RoboDK station: CSU Expo Station.rdk

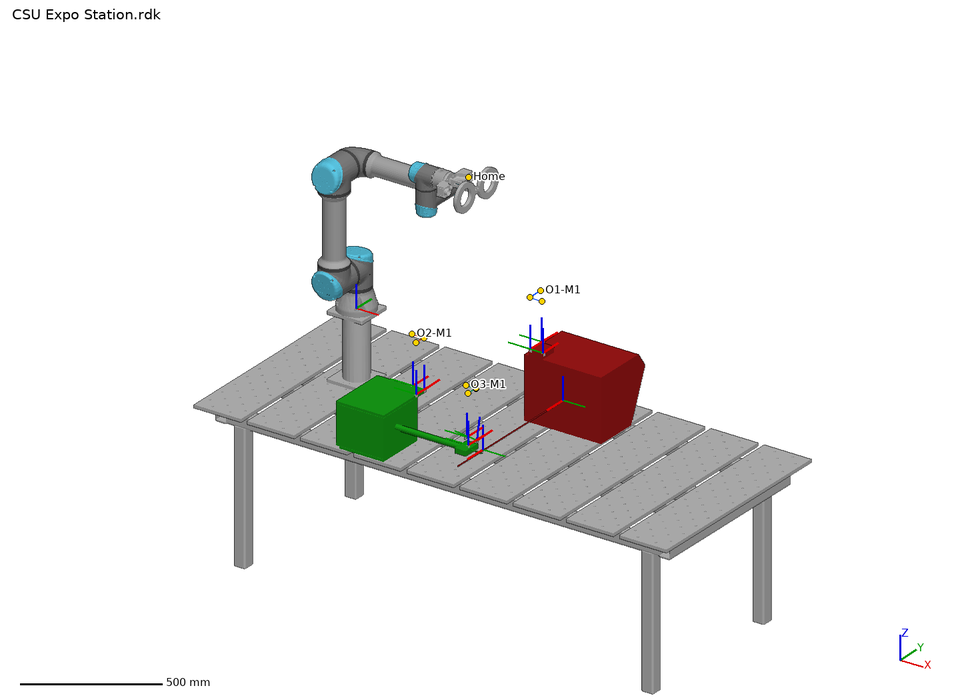
[picture v0: the station drawn from its stored meshes, robots at their saved joint values, targets as dots, program paths as lines]
Station CSU Expo Station (saved by RoboDK 5.0.1). Poses are relative to the parent item; angles as X-Y-Z fixed-axis rotations.
  - object Welding Table at (-1600, 2170, 0) mm, rotated rx 90 ry 0 rz 0 deg, size 2032 x 628.6 x 889 mm, geometry from Welding Table.STEP
  - object Tower_V4.1 (2) at (-1504.7, 555.63, 733.6) mm, size 152.4 x 152.4 x 279.4 mm, geometry from Tower_V4.1 (2).STEP
  - object X-Ray Box (3) at (-679.2, 641.63, 724.08) mm, rotated rx 0 ry 0 rz -90 deg, size 914.8 x 330 x 284 mm, geometry from X-Ray Box (3).STEP
  - object Kappa Expo (1) at (-1059.7, 166.63, 724.08) mm, rotated rx 0 ry 0 rz -90 deg, size 256 x 575.5 x 181.2 mm, geometry from Kappa Expo (1).STEP
  - frame UR5e Base at (-1504.7, 555.63, 1013) mm
    - robot UR5e: 6 axes, payload 5 kg, reach 850 mm, repeatability 0.03 mm, weight 18.4 kg
        modified DH rows (alpha deg, a mm, theta deg, d mm): 0, 0, 0, 162.5; 90, 0, 180, 0; 0, 425, 0, 0; 0, 392.25, 0, 133.3; -90, 0, 0, 99.7; 90, 0, 180, 99.6
        joint limits [-360, -360, -360, -360, -360, -360] to [360, 360, 360, 360, 360, 360]; home [0, -90, -90, 0, 90, 0]; saved at [0, -90, -90, 0, 90, 0]
      - tool Left Camera, TCP at (-69.39, 0, 34.3) mm, size 256 x 114.2 x 122.3 mm
      - tool Right Camera, TCP at (69.39, 0, 34.3) mm
    - target Home (Cartesian target) at (526.15, -63.91, 687.2) mm, rotated rx -90 ry 0 rz -90 deg; joints [0, -90, -90, 0, 90, 0] of UR5e
    - target O1-M1 (Cartesian target) at (682, 157, 198.5) mm, rotated rx 180 ry 0 rz -90 deg; joints [18.498, -122.802, -85.726, -61.472, 90.002, 18.498] of UR5e
    - target O1-M2 (Cartesian target) at (682, 89, 198.5) mm, rotated rx -180 ry 0 rz -90 deg; joints [12.914, -122.158, -86.796, -61.046, 89.997, 12.914] of UR5e
    - target O1-M3 (Cartesian target) at (735, 89, 198.5) mm, rotated rx 180 ry 0 rz -90 deg; joints [11.974, -128.74, -75.588, -65.672, 89.998, 11.974] of UR5e
    - target O2-M1 (Cartesian target) at (392, -217.96, 96) mm, rotated rx 180 ry 0 rz -90 deg; joints [-20.326, -111.217, -125.737, -33.048, 90.003, -20.326] of UR5e
    - target O2-M2 (Cartesian target) at (442, -217.96, 96) mm, rotated rx 180 ry 0 rz -90 deg; joints [-18.383, -115.073, -118.98, -35.949, 90, -18.383] of UR5e
    - target O2-M3 (Cartesian target) at (442, -267.96, 96) mm, rotated rx 180 ry 0 rz -90 deg; joints [-23.481, -117.773, -114.117, -38.113, 89.999, -23.481] of UR5e
    - target O3-M1 (Cartesian target) at (723, -359.5, 44.31) mm, rotated rx 180 ry 0 rz -90 deg; joints [-21.553, -153.256, -53.33, -63.416, 90, -21.553] of UR5e
    - target O3-M2 (Cartesian target) at (765, -359.5, 44.31) mm, rotated rx 180 ry 0 rz -90 deg; joints [-20.535, -159.517, -40.305, -70.18, 90.001, -20.535] of UR5e
    - target O3-M3 (Cartesian target) at (765, -409.5, 44.31) mm, rotated rx 180 ry 0 rz -90 deg; joints [-23.553, -165.459, -27.955, -76.587, 90.001, -23.553] of UR5e
    - target Target 11 (Cartesian target) at (765.02, -359.5, 46.15) mm, rotated rx -180 ry 0 rz -89.99 deg; joints [-20.534, -159.392, -40.279, -70.329, 90.004, -20.543] of UR5e
  - Python program Prog1 (listed below)
  - program OB1 (6 instructions, listed below)
  - program OB2 (6 instructions, listed below)
  - program OB3 (6 instructions, listed below)
  - program hOME (4 instructions, listed below)
  - Python program Prog6 (listed below)
  - frame Specimen at (-689.2, 166.63, 844.08) mm, rotated rx 0 ry 0 rz -90 deg
  - frame O1-M1 at (-819.7, 715.63, 1010.08) mm, rotated rx 0 ry 0 rz 90 deg
    - object O1-M1 at (3, -3, 0) mm, rotated rx 0 ry 0 rz 90 deg, size 10 x 10 x 10 mm, geometry from Fiducial Edge (1).STEP
  - frame O1-M2 at (-819.7, 644.63, 1010.08) mm, rotated rx 0 ry 0 rz 90 deg
    - object O1-M2 at (0, -3, 0) mm, rotated rx 0 ry 0 rz 90 deg, size 10 x 10 x 10 mm, geometry from Fiducal Corner.STEP
  - frame O1-M3 at (-766.7, 644.63, 1010.08) mm, rotated rx 0 ry 0 rz 90 deg
    - object O1-M3 at (0, -3, 0) mm, rotated rx 0 ry 0 rz -90 deg, size 10 x 10 x 10 mm, geometry from Fiducial Edge (1).STEP
  - frame O2-M1 at (-1109.7, 337.67, 907.33) mm, rotated rx 0 ry 0 rz 90 deg
    - object O2-M1 at (0, 3, 0) mm, size 10 x 10 x 10 mm, geometry from Fiducial Edge (1).STEP
  - frame O2-M2 at (-1059.7, 337.67, 907.33) mm, rotated rx 0 ry 0 rz 90 deg
    - object O2-M2 at (0, 3, 0) mm, rotated rx 0 ry 0 rz -180 deg, size 10 x 10 x 10 mm, geometry from Fiducal Corner.STEP
  - frame O2-M3 at (-1059.7, 287.67, 907.33) mm, rotated rx 0 ry 0 rz 90 deg
    - object O2-M3 at (0, 3, 0) mm, rotated rx 0 ry 0 rz -90 deg, size 10 x 10 x 10 mm, geometry from Fiducial Edge (1).STEP
  - frame O3-M1 at (-778.7, 196.13, 856.08) mm, rotated rx 0 ry 0 rz 90 deg
    - object O3-M1 at (0, 3, 0) mm, rotated rx 0 ry 0 rz 90 deg, size 10 x 10 x 10 mm, geometry from Fiducial Edge (1).STEP
  - frame O3-M2 at (-735.04, 196.13, 855.98) mm, rotated rx 6.36 ry -0.02 rz 90.28 deg
    - object O3-M2 at (0, 3, 0) mm, rotated rx 0 ry 0 rz -180 deg, size 10 x 10 x 10 mm, geometry from Fiducal Corner.STEP
  - frame O3-M3 at (-736.7, 146.13, 856.08) mm, rotated rx 0 ry 0 rz 90 deg
    - object O3-M3 at (0, 3, 0) mm, rotated rx 0 ry 0 rz -90 deg, size 10 x 10 x 10 mm, geometry from Fiducial Edge (1).STEP
  - frame X-Ray Outlet at (-679.2, 642.63, 849.08) mm, rotated rx 0 ry 0 rz -90 deg
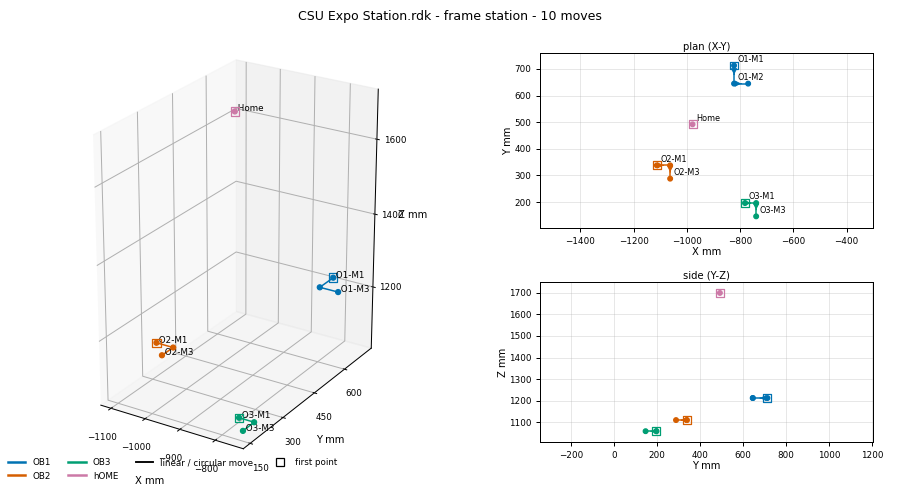
[picture p0: tool path of CSU Expo Station.rdk in frame station, 10 of 10 moves have a stored position in this frame; points joined in program order, loops and branches not executed]

--- Python program Prog1 ---
from robolink import *    # RoboDK's API
from robodk import *      # Math toolbox for robots
import logging
import sys, time, math

RDK = robolink.Robolink()

# OpenCV is an open source Computer Vision toolkit, which you can use to filter and analyse images
robolink.import_install('cv2', 'opencv-contrib-python', RDK)
robolink.import_install('numpy', RDK)

sys.path.insert(1, r'C:\Users\PoThe\OneDrive\Desktop\VimbaPython_Source')
import numpy as np
import cv2 as cv
import cv2
from cv2 import VideoCapture, aruco
from vimba import *
import measure_class

logging.basicConfig(filename="TestRun.log",level=logging.INFO,filemode='w')

calib_path  = r'C:\Users\PoThe\OneDrive\Desktop\VimbaPython_Source'
camera_matrix   = np.loadtxt(calib_path+'\cameraMatrix.txt', delimiter=',')
camera_distortion   = np.loadtxt(calib_path+'\cameraDistortion.txt', delimiter=',')

marker_actual = 6 #[mm]

marker_size  =  marker_actual/10 # how it will be processed [cm]

# Define Robot:
robot = RDK.Item('UR5e', ITEM_TYPE_ROBOT)
O1M1 = RDK.Item('O1-M1',ITEM_TYPE_OBJECT)

O1_M1_xyz = list()

O1_M1 = measure_class.measure(0,0,0,0)
O1M1_Xray = (73, -140.5, 161.00)
def offset(y,z):
    osy = y+30
    osz = z+6
    return osy, osz

TCP = robot.Pose()
O1_M1.measuring(marker_size, calib_path, camera_matrix, camera_distortion)
cv2.destroyAllWindows()
x = -O1_M1.x
O1_M1_xyz.append(x)
O1_M1_xyz.append(O1_M1.y)
O1_M1_xyz.append(O1_M1.z)

O1M1_Base = TCP*transl(O1_M1_xyz)
x,y,z,rx,ry,rz = Pose_2_TxyzRxyz(O1M1_Base)
y,z = offset(y,z)
O1M1_Base = TxyzRxyz_2_Pose([x,y,z,rx,ry,rz])

O1_X1 = O1M1_Base*transl(O1M1_Xray)
x1,y1,z1,rx1,ry1,rz1 = Pose_2_TxyzRxyz(O1_X1)

logging.info("Marker 1 to base: %s", O1M1_Base)

logging.info("X-ray to base: %s", O1_X1)

--- program OB1 (robot UR5e) ---
  Set Ref.: UR5e Base
  Set Tool: Left Camera
  Set speed (200.0 mm/s)
  MoveL (O1-M1)
  MoveL (O1-M2)
  MoveL (O1-M3)

--- program OB2 (robot UR5e) ---
  Set Ref.: UR5e Base
  Set Tool: Left Camera
  Set speed (200.0 mm/s)
  MoveL (O2-M1)
  MoveL (O2-M2)
  MoveL (O2-M3)

--- program OB3 (robot UR5e) ---
  Set Ref.: UR5e Base
  Set Tool: Left Camera
  Set speed (200.0 mm/s)
  MoveL (O3-M1)
  MoveL (O3-M2)
  MoveL (O3-M3)

--- program hOME (robot UR5e) ---
  Set Ref.: UR5e Base
  Set Tool: Left Camera
  Set speed (100.0 mm/s)
  MoveL (Home)

--- Python program Prog6 ---
from robolink import *    # RoboDK's API
from robodk import *      # Math toolbox for robots
import logging
import sys, time, math

RDK = robolink.Robolink()

# OpenCV is an open source Computer Vision toolkit, which you can use to filter and analyse images
robolink.import_install('cv2', 'opencv-contrib-python', RDK)
robolink.import_install('numpy', RDK)

sys.path.insert(1, r'C:\Users\PoThe\OneDrive\Desktop\VimbaPython_Source')
import numpy as np
import cv2 as cv
import cv2
from cv2 import VideoCapture, aruco
from vimba import *
import measure_class

logging.basicConfig(filename="TestRun.log",level=logging.INFO,filemode='w')

calib_path  = r'C:\Users\PoThe\OneDrive\Desktop\VimbaPython_Source'
camera_matrix   = np.loadtxt(calib_path+'\cameraMatrix.txt', delimiter=',')
camera_distortion   = np.loadtxt(calib_path+'\cameraDistortion.txt', delimiter=',')

marker_actual = 6 #[mm]

marker_size  =  marker_actual/10 # how it will be processed [cm]

# Program example:
robot = RDK.Item('UR5e', ITEM_TYPE_ROBOT)
Home = RDK.Item('Home', ITEM_TYPE_TARGET)
O1M1 = RDK.Item('O1-M1', ITEM_TYPE_TARGET)
O1M2 = RDK.Item('O1-M2', ITEM_TYPE_TARGET)
O1M3 = RDK.Item('O1-M3', ITEM_TYPE_TARGET)
O2M1 = RDK.Item('O2-M1', ITEM_TYPE_TARGET)
O2M2 = RDK.Item('O2-M2', ITEM_TYPE_TARGET)
O2M3 = RDK.Item('O2-M3', ITEM_TYPE_TARGET)
O3M1 = RDK.Item('O3-M1', ITEM_TYPE_TARGET)
O3M2 = RDK.Item('O3-M2', ITEM_TYPE_TARGET)
O3M3 = RDK.Item('O3-M3', ITEM_TYPE_TARGET)

#ArUco Markers
O1_M1 = measure_class.measure(0,0,0,0)
O1_M2 = measure_class.measure(0,0,0,0)
O1_M3 = measure_class.measure(0,0,0,0)
O2_M1 = measure_class.measure(0,0,0,0)
O2_M2 = measure_class.measure(0,0,0,0)
O2_M3 = measure_class.measure(0,0,0,0)
O3_M1 = measure_class.measure(0,0,0,0)
O3_M2 = measure_class.measure(0,0,0,0)
O3_M3 = measure_class.measure(0,0,0,0)

#xyz coordinates
O1_M1_xyz = list()
O1_M2_xyz = list()
O1_M3_xyz = list()
O2_M1_xyz = list()
O2_M2_xyz = list()
O2_M3_xyz = list()
O3_M1_xyz = list()
O3_M2_xyz = list()
O3_M3_xyz = list()

#xyz of the reference frame 'X-ray Output' with respect to marker locations
#O1M1_Xray = (140.5, -71.00, -161.00)
O1M1_Xray = (73, -140.5, 161.00)
O1M2_Xray = (-2, -140.5, 161.00)
O1M3_Xray = (-2, -87.500, 161.00)

O2M1_Xray = (-304.960, -433.500, 58.250)
O2M2_Xray = (-304.960, -383.500, 58.250)
O2M3_Xray = (-354.960, -383.500, 58.250)

#xyz of the reference frame 'Specimen' with respect to marker locations
O3M1_Spec = (-29.5, -89.500, 12.000)
O3M2_Spec = (-29.504, -45.838, 11.908)
O3M3_Spec = (-20.500, -47.50, 12.00)

XR_xlist = list()
XR_ylist = list()
XR_zlist = list()
S_xlist = list()
S_ylist = list()
S_zlist = list()

def offset(y,z):
    osy = y+30
    osz = z+6
    return osy, osz

def home():
    robot.MoveL(Home)

def object1():

#MARKER 1
    #--------------------------------------------------------------------------------------------------------------------
    robot.MoveL(O1M1)
    TCP = robot.Pose()
    O1_M1.measuring(marker_size, calib_path, camera_matrix, camera_distortion)
    cv2.destroyAllWindows()
    x = -O1_M1.x
    O1_M1_xyz.append(x)
    O1_M1_xyz.append(O1_M1.y)
    O1_M1_xyz.append(O1_M1.z)

    O1M1_Base = TCP*transl(O1_M1_xyz)
    x,y,z,rx,ry,rz = Pose_2_TxyzRxyz(O1M1_Base)
    y,z = offset(y,z)
    O1M1_Base = TxyzRxyz_2_Pose([x,y,z,rx,ry,rz])

    O1_X1 = O1M1_Base*transl(O1M1_Xray)
    x1,y1,z1,rx1,ry1,rz1 = Pose_2_TxyzRxyz(O1_X1)
    XR_xlist.append(x1)
    XR_ylist.append(y1)
    XR_zlist.append(z1)
    logging.info("Marker 1 to base: %s", O1M1_Base)
    #--------------------------------------------------------------------------------------------------------------------

#MARKER 2
    #--------------------------------------------------------------------------------------------------------------------
    robot.MoveL(O1M2)
    TCP = robot.Pose()
    O1_M2.measuring(marker_size, calib_path, camera_matrix, camera_distortion)
    cv2.destroyAllWindows()
    x = -O1_M2.x
    O1_M2_xyz.append(x)
    O1_M2_xyz.append(O1_M2.y)
    O1_M2_xyz.append(O1_M2.z)

    O1M2_Base = TCP*transl(O1_M2_xyz)
    x,y,z,rx,ry,rz = Pose_2_TxyzRxyz(O1M2_Base)
    y,z = offset(y,z)
    O1M2_Base = TxyzRxyz_2_Pose([x,y,z,rx,ry,rz])

    O1_X2 = O1M2_Base*transl(O1M2_Xray)
    x2,y2,z2,rx2,ry2,rz2 = Pose_2_TxyzRxyz(O1_X2)
    XR_xlist.append(x2)
    XR_ylist.append(y2)
    XR_zlist.append(z2)
    logging.info("Marker 2 to base: %s", O1M2_Base)
    #--------------------------------------------------------------------------------------------------------------------

#MARKER 3
    #--------------------------------------------------------------------------------------------------------------------
    robot.MoveL(O1M3)
    TCP = robot.Pose()
    O1_M3.measuring(marker_size, calib_path, camera_matrix, camera_distortion)
    cv2.destroyAllWindows()
    x = -O1_M3.x
    O1_M3_xyz.append(x)
    O1_M3_xyz.append(O1_M3.y)
    O1_M3_xyz.append(O1_M3.z)

    O1M3_Base = TCP*transl(O1_M3_xyz)
    #logging.info("Marker ID: %s \nCamera Pos w/ respect to marker: x = %2.3f, y = %2.3f, z = %2.3f \nMarker matrix w/respect to base: %s\n", O1_M3.markerid[0], O1_M3.x, O1_M3.y, O1_M3.z, O1M3_Base)
    x,y,z,rx,ry,rz = Pose_2_TxyzRxyz(O1M3_Base)
    y,z = offset(y,z)
    O1M3_Base = TxyzRxyz_2_Pose([x,y,z,rx,ry,rz])
    logging.info("Marker 3 to base: %s", O1M3_Base)

    O1_X3 = O1M3_Base*transl(O1M3_Xray)
    x3,y3,z3,rx3,ry3,rz3 = Pose_2_TxyzRxyz(O1_X3)
    XR_xlist.append(x3)
    XR_ylist.append(y3)
    XR_zlist.append(z3)
    #--------------------------------------------------------------------------------------------------------------------

    logging.info("X-ray coordinates with respect to Base: \nPosition 1: %s \nPosition 2: %s \nPosition 3: %s",O1_X1, O1_X2, O1_X3)

def object2():
#MARKER 4
    #------------------------------------------------------------------------------------------------------------------
    robot.MoveL(O2M1)
    TCP = robot.Pose()
    O2_M1.measuring(marker_size, calib_path, camera_matrix, camera_distortion)
    cv2.destroyAllWindows()
    x = -O2_M1.x
    O2_M1_xyz.append(x)
    O2_M1_xyz.append(O2_M1.y)
    O2_M1_xyz.append(O2_M1.z)
    O2M1_Base = TCP*transl(O2_M1_xyz)

    O2M1_Base = TCP*transl(O2_M1_xyz)
    x,y,z,rx,ry,rz = Pose_2_TxyzRxyz(O2M1_Base)
    #y,z = offset(y,z)
    O2M1_Base = TxyzRxyz_2_Pose([x,y,z,rx,ry,rz])


    O2_X1 = O2M1_Base*transl(O2M1_Xray)
    x4,y4,z4,rx4,ry4,rz4 = Pose_2_TxyzRxyz(O2_X1)
    XR_xlist.append(x4)
    XR_ylist.append(y4)
    XR_zlist.append(z4)
    logging.info("Marker 4 with respect to base: %s", O2M1_Base)

#MARKER 5
    #----------------------------------------------------------------------------------------------------------------------
    robot.MoveL(O2M2)
    TCP = robot.Pose()
    O2_M2.measuring(marker_size, calib_path, camera_matrix, camera_distortion)
    cv2.destroyAllWindows()
    x = -O2_M2.x
    O2_M2_xyz.append(x)
    O2_M2_xyz.append(O2_M2.y)
    O2_M2_xyz.append(O2_M2.z)
    O2M2_Base = TCP*transl(O2_M2_xyz)

    O2M2_Base = TCP*transl(O2_M2_xyz)
    x2,y2,z2,rx2,ry2,rz2 = Pose_2_TxyzRxyz(O2M2_Base)
    #y2,z2 = offset(y2,z2)
    O2M2_Base = TxyzRxyz_2_Pose([x2,y2,z2,rx2,ry2,rz2])

    logging.info("Marker 5 with respect to base: %s", O2M2_Base)
    O2_X2 = O2M2_Base*transl(O2M2_Xray)
    x5,y5,z5,rx5,ry5,rz5 = Pose_2_TxyzRxyz(O2_X2)
    XR_xlist.append(x5)
    XR_ylist.append(y5)
    XR_zlist.append(z5)

    #-------------------------------------------------------------------------------------------------------------------------------

#MARKER 6
    #-----------------------------------------------------------------------------------------------------------------------------
    robot.MoveL(O2M3)
    TCP = robot.Pose()
    O2_M3.measuring(marker_size, calib_path, camera_matrix, camera_distortion)
    cv2.destroyAllWindows()

    x = -O2_M3.x
    O2_M3_xyz.append(x)
    O2_M3_xyz.append(O2_M3.y)
    O2_M3_xyz.append(O2_M3.z)
    O2M3_Base = TCP*transl(O2_M3_xyz)

    O2M3_Base = TCP*transl(O2_M3_xyz)
    x3,y3,z3,rx3,ry3,rz3 = Pose_2_TxyzRxyz(O2M3_Base)
    y3,z3 = offset(y3,z3)
    O2M3_Base = TxyzRxyz_2_Pose([x3,y3,z3,rx3,ry3,rz3])
    #logging.info("Marker with respect to base: %s",O2M3_Base)
    O2_X3 = O2M3_Base*transl(O2M3_Xray)
    x6,y6,z6,rx6,ry6,rz6 = Pose_2_TxyzRxyz(O2_X3)
    XR_xlist.append(x6)
    XR_ylist.append(y6)
    XR_zlist.append(z6)
    logging.info("Marker 6 with respect to base: %s", O2M3_Base)
    #----------------------------------------------------------------------------------------------------------------------------------

    xavg = sum(XR_xlist[0:])/len(XR_xlist)
    yavg = sum(XR_ylist[0:])/len(XR_ylist)
    zavg = sum(XR_zlist[0:])/len(XR_zlist)

    XR = TxyzRxyz_2_Pose([xavg,yavg,zavg,0,0,0])

    logging.info("X-ray coordinates with respect to Base: \nPosition 4: %s \nPosition 5: %s \nPosition 6: %s",O2_X1, O2_X2, O2_X3)
    logging.info("X-ray coordinates with respect to base: %s",XR)



def object3():
#MARKER 7
    #----------------------------------------------------------------------------------------
    robot.MoveL(O3M1)
    TCP = robot.Pose()
    O3_M1.measuring(marker_size, calib_path, camera_matrix, camera_distortion)
    cv2.destroyAllWindows()
    x = -O3_M1.x
    O3_M1_xyz.append(O3_M1.x)
    O3_M1_xyz.append(O3_M1.y)
    O3_M1_xyz.append(O3_M1.z)
    O3M1_Base = TCP*transl(O3_M1_xyz)
    #logging.info("Marker ID: %s \nCamera Pos w/ respect to marker: x = %2.3f, y = %2.3f, z = %2.3f \nMarker matrix w/respect to base: %s\n", O3_M1.markerid[0], O3_M1.x, O3_M1.y, O3_M1.z, O3M1_Base)
    O3_S1 = O3M1_Base*transl(O3M1_Spec)
    Sx1,Sy1,Sz1,Srx1,Sry1,Srz1 = Pose_2_TxyzRxyz(O3_S1)
    S_xlist.append(Sx1)
    S_ylist.append(Sy1)
    S_zlist.append(Sz1)
    logging.info("Marker 7 with respect to base: %s", O3M1_Base)
    #---------------------------------------------------------------------------------

#MARKER 8
    #-------------------------------------------------------------------------------------
    robot.MoveL(O3M2)
    TCP = robot.Pose()
    O3_M2.measuring(marker_size, calib_path, camera_matrix, camera_distortion)
    cv2.destroyAllWindows()

    x = -O3_M2.x
    O3_M2_xyz.append(O3_M2.x)
    O3_M2_xyz.append(O3_M2.y)
    O3_M2_xyz.append(O3_M2.z)
    O3M2_Base = TCP*transl(O3_M2_xyz)
    #logging.info("Marker ID: %s \nCamera Pos w/ respect to marker: x = %2.3f, y = %2.3f, z = %2.3f \nMarker matrix w/respect to base: %s\n", O3_M2.markerid[0], O3_M2.x, O3_M2.y, O3_M2.z, O3M2_Base)
    O3_S2 = O3M2_Base*transl(O3M2_Spec)
    Sx2,Sy2,Sz2,Srx2,Sry2,Srz2 = Pose_2_TxyzRxyz(O3_S2)
    S_xlist.append(Sx2)
    S_ylist.append(Sy2)
    S_zlist.append(Sz2)
    logging.info("Marker 8 with respect to base: %s", O3M2_Base)
    #---------------------------------------------------------------------------------------

#MARKER 9
    #------------------------------------------------------------------------------------------
    robot.MoveL(O3M3)
    TCP = robot.Pose()
    O3_M3.measuring(marker_size, calib_path, camera_matrix, camera_distortion)
    cv2.destroyAllWindows()
    x = -O3_M3.x
    O3_M3_xyz.append(O3_M3.x)
    O3_M3_xyz.append(O3_M3.y)
    O3_M3_xyz.append(O3_M3.z)
    O3M3_Base = TCP*transl(O3_M3_xyz)
    #logging.info("Marker ID: %s \nCamera Pos w/ respect to marker: x = %2.3f, y = %2.3f, z = %2.3f \nMarker matrix w/respect to base: %s\n", O3_M3.markerid[0], O3_M3.x, O3_M3.y, O3_M3.z, O3M3_Base)
    O3_S3 = O3M3_Base*transl(O3M3_Spec)
    Sx3,Sy3,Sz3,Srx3,Sry3,Srz3 = Pose_2_TxyzRxyz(O3_S3)
    S_xlist.append(Sx3)
    S_ylist.append(Sy3)
    S_zlist.append(Sz3)
    logging.info("Marker 9 with respect to base: %s", O3M3_Base)
    #----------------------------------------------------------------------------------------

    Sxavg = sum(S_xlist[0:])/len(S_xlist)
    Syavg = sum(S_ylist[0:])/len(S_ylist)
    Szavg = sum(S_zlist[0:])/len(S_zlist)

    S = TxyzRxyz_2_Pose([Sxavg,Syavg,Szavg,0,0,0])
    logging.info("Specimen coordinates with respect to Base: \nPosition 1: %s \nPosition 2: %s \nPosition 3: %s",O3_S1, O3_S2, O3_S3)
    logging.info("Specimen coordinates with respect to base: %s",S)

#main
robot.setPoseFrame(robot.PoseFrame())
robot.setPoseTool(robot.PoseTool())
#robot.setRounding(10)  # Set the rounding parameter (Also known as: CNT, APO/C_DIS, ZoneData, Blending radius, cornering, ...)
robot.setAcceleration(1000)
robot.setSpeed(800)#set linear speed to 200mm/s

home()
tic = time.perf_counter()
object1()
object2()
object3()
tac = time.perf_counter()
home()
toe = tac - tic
logging.info('total runtime: %s',toe)
